{attribute 'GeneratedUsingTerminal: EL9180--0000'}
{attribute addProperty BoxType "EL9180--0000"}
{attribute addProperty Description "EL9180 Potential Connection, 2 x 24-230V, 2 x PE"}
{attribute addProperty Physics "KK"}
{attribute addProperty Id "EL9180"}
{attribute addProperty CRC "2333413004"}
{attribute addProperty Size "0"}
TYPE EL9180_8B150E8C EXTENDS EtcSlaveTerminalBase_947E5A46 :
STRUCT
END_STRUCT
END_TYPE

(* stored: Version 1.2.0.0, ProductVersion 3.1.4024.11
   DUT EL9180_8B150E8C: Id {d5d90ef4-6872-41a8-824c-fa53210b9ade} *)
